/// Data of one tracking zone
TYPE ST_WindowTrackingZone :
(************************************************************************************** 
* 	Application 		: BoxControl Framework 
* 	Revision 			: $Revision: 408723 $ 
* 	Revision date 		: $Date: 2018-06-27 13:49:08 +0200 (Wed, 27 Jun 2018) $ 
* 	Last changed by 	: $Author: b7bolm $ 
* 	URL 				: $URL: http://almscdc.swisslog.com/repo/SWPD/Development/BoxControlFramework/21_Projects/BCF_2.0/trunk/BCF/BCF/JumpStart/20_Product/10_App/12_E_Functions/10_Lib/10_Conv/FB_FunctionList.TcPOU $ 
* ------------------------------------------------------------------------------------ 
* 	© Swisslog AG 
* 	Swisslog is not liable for any usage of this source code that is not agreed 
* 	on between Swisslog and the other party. The mandatory legal liability remains 
* 	unaffected. 
* ------------------------------------------------------------------------------------ 
* 	Revision History: 
* 
* 	VERSION 		DATE 			INITIALS 			DESCRIPTION 
* 	0.1 			24.08.2018 		ahe 				First implementation
* 
**************************************************************************************)
STRUCT
	Used					: BOOL;
	ActionId				: INT;
	ZoneLength				: UINT;
	ZoneStartWindowIndex	: UINT;
	ZoneEndWindowIndex		: UINT;
	ZoneStartPosition		: UDINT;
	ZoneEndPosition			: UDINT;
	TU_StartWindowIndex		: UINT;
	TU_EndWindowIndex		: UINT;
	TU_Present				: BOOL;
	TU_Index				: DINT;
	Flush					: BOOL; 
	InhibitShifting			: BOOL;
	PositionToLive			: UDINT;
	iActionListener			: I_TrackingActionListener;
END_STRUCT
END_TYPE

(* stored: Version 1.1.0.1, ProductVersion 3.1.4022.12
   DUT ST_WindowTrackingZone: Id {45a7366d-5411-47c4-9274-7438f90fd003} *)
